{attribute 'no_check'}
//EL3356 load cell analysis (resistor bridge) process image
//Mode of operation = Standard (Real or INT32)
FUNCTION_BLOCK EL3356 EXTENDS EcSlaveInfoDataExt
VAR_INPUT
//RMB Control
	StartCalib										AT  %Q* : 	BOOL; 
	DisableCalib									AT  %Q* : 	BOOL;
	InputFreeze										AT  %Q* : 	BOOL;
	SampleMode										AT  %Q* : 	BOOL; //1=High speed and low latency / only on EL3356-0010
	Tara											AT  %Q* : 	BOOL;				
END_VAR                     			    					
VAR_OUTPUT                      					
//RMB Status
	Overrange										AT  %I*	:	BOOL;
	DataInvalid										AT  %I*	:	BOOL;
	Error											AT  %I*	:	BOOL;
	CalibInProgress									AT  %I*	:	BOOL;
	SteadyState										AT  %I*	:	BOOL;
	SyncError										AT  %I*	:	BOOL;
	TxPDOToggle										AT  %I* : 	BOOL;
	
//RMB Value
	InReal											AT  %I* : 	REAL; //RMP Value Real 32		
	InInt32											AT  %I* : 	DINT; //RMB Value INT32
END_VAR
VAR
END_VAR

(* EL3356 IOs											             	 		*)
(********************************************************************************)

(* ******************************************************************************)
	Super^();
(********************************************************************************)

{attribute 'monitoring' := 'call'}
PROPERTY PUBLIC inError : BOOL
GET
inError													:= Error OR SyncError OR WcState OR InfoDataState <> Tc2_EtherCAT.EC_DEVICE_STATE_OP;
END_GET
END_PROPERTY

{attribute 'monitoring' := 'call'}
PROPERTY PUBLIC Q : LREAL
GET
IF InInt32 <> 0
THEN
	Q 														:= TO_LREAL(InInt32);
ELSE
	Q 														:= TO_LREAL(InReal);
END_IF
END_GET
END_PROPERTY

{attribute 'monitoring' := 'call'}
PROPERTY Q_GramToNewton : LREAL
GET
Q_GramToNewton := GF_TO_N(Q);
END_GET
END_PROPERTY

{attribute 'monitoring' := 'call'}
PROPERTY Q_NewtonToGram : LREAL
GET
Q_NewtonToGram := N_TO_GF(Q);
END_GET
END_PROPERTY

END_FUNCTION_BLOCK

(* stored: Version 1.1.0.1, ProductVersion 3.1.4024.12
   POU EL3356: Id {cf7101d6-3b87-4f3e-babb-afb08e318558}, SpecialFunc None
   Property inError: Id {d75d9581-3d2a-4fa5-85dd-9ce5affabb4e}
   Get Get: Id {ed613275-0d58-4a90-aa81-b36ac781c140}
   Property Q: Id {651deb2c-dafe-4190-bf0f-b5537ac8439b}
   Get Get: Id {be13110d-4495-41ad-970b-0826e7efded5}
   Property Q_GramToNewton: Id {1984eb02-6b8d-48f3-9df5-352bd4b92454}
   Get Get: Id {37f5f8a4-b6b0-4bdd-82a4-ac3835a79bb6}
   Property Q_NewtonToGram: Id {fd191490-ab0a-446e-9b17-fdb91b0fe8ff}
   Get Get: Id {40a8fc4a-85e3-4271-9e20-c75f3172a67b} *)
